// TIA Portal V20 export
TYPE "typeEm2MonitoringCmStatus"
// stored: Access Published, Namespace Unit1
   STRUCT
      electrodeFixRightTop { ExternalWritable := 'False'} : "LBC_typeTwoWayActuatorControlNodeMonitoring";
      electrodeFixRightBottom { ExternalWritable := 'False'} : "LBC_typeTwoWayActuatorControlNodeMonitoring";
      electrodeFixLeftTop { ExternalWritable := 'False'} : "LBC_typeTwoWayActuatorControlNodeMonitoring";
      electrodeFixLeftBottom { ExternalWritable := 'False'} : "LBC_typeTwoWayActuatorControlNodeMonitoring";
      electrodeFixLeftTopLift { ExternalWritable := 'False'} : "LBC_typeTwoWayActuatorControlNodeMonitoring";
      electrodeFixLeftBottomLift { ExternalWritable := 'False'} : "LBC_typeTwoWayActuatorControlNodeMonitoring";
      uwSplicerVacRightTop { ExternalWritable := 'False'} : "LBC_typeTwoWayActuatorControlNodeMonitoring";
      uwSplicerVacRightBottom { ExternalWritable := 'False'} : "LBC_typeTwoWayActuatorControlNodeMonitoring";
      uwSplicerVacLeftTop { ExternalWritable := 'False'} : "LBC_typeTwoWayActuatorControlNodeMonitoring";
      uwSplicerVacLeftBottom { ExternalWritable := 'False'} : "LBC_typeTwoWayActuatorControlNodeMonitoring";
      electrodeCutter { ExternalWritable := 'False'} : "LBC_typeTwoWayActuatorControlNodeMonitoring";
      splicingLeftMover { ExternalWritable := 'False'} : "LBC_typeTwoWayActuatorControlNodeMonitoring";
      splicingRightMover { ExternalWritable := 'False'} : "LBC_typeTwoWayActuatorControlNodeMonitoring";
      electrodeLeftHolder { ExternalWritable := 'False'} : "LBC_typeTwoWayActuatorControlNodeMonitoring";
      electrodeRightHolder { ExternalWritable := 'False'} : "LBC_typeTwoWayActuatorControlNodeMonitoring";
      tapeLoadingTurn { ExternalWritable := 'False'} : "LBC_typeTwoWayActuatorControlNodeMonitoring";
      tapeAttachUnit { ExternalWritable := 'False'} : "LBC_typeTwoWayActuatorControlNodeMonitoring";
      uwSplicerTapeVac { ExternalWritable := 'False'} : "LBC_typeTwoWayActuatorControlNodeMonitoring";
      stopper { ExternalWritable := 'False'} : "LBC_typeTwoWayActuatorControlNodeMonitoring";
      supportTransfer { ExternalWritable := 'False'} : "LBC_typeTwoWayActuatorControlNodeMonitoring";
      supportShaftLift { ExternalWritable := 'False'} : "LBC_typeTwoWayActuatorControlNodeMonitoring";
      frameCover { ExternalWritable := 'False'} : "LBC_typeTwoWayActuatorControlNodeMonitoring";
   END_STRUCT;
END_TYPE
